TYPE ValueArray :
STRUCT
	q1		: ARRAY[0..7] OF BYTE;
	q2		: ARRAY[0..7] OF BYTE;
	q3		: ARRAY[0..7] OF BYTE;
	q4		: ARRAY[0..7] OF BYTE;
	q5		: ARRAY[0..7] OF BYTE;
	q6		: ARRAY[0..7] OF BYTE;
END_STRUCT
END_TYPE

(* stored: Version 1.1.0.1
   DUT ValueArray: Id {87ac232e-b4e8-475b-be64-2ab880a62e67} *)
